Fanuc KAREL source: SET_REAL_REG.kl

PROGRAM T
%NOLOCKGROUP
VAR
 v0 : INTEGER
 v1 : REAL
 v2 : INTEGER
BEGIN
 SET_REAL_REG(v0, v1, v2)
END T
